FUNCTION_BLOCK FB_RecipeAnalogInputControlSequencer
VAR_INPUT
	rampTime: UINT;
END_VAR
VAR_IN_OUT
	rRecipe: ARRAY[1..GVL_IO.nNumController] OF REAL;
END_VAR
VAR
	i: INT;
END_VAR

FOR i:= 1 TO GVL_IO.nNumMFC DO
	GVL_IO.aController[i].input.restart := TRUE;
	GVL_IO.aController[i].input.rampTime := rampTime; 
	GVL_IO.aController[i].input.targetValue := rRecipe[i] / GVL_IO.aMaxValueController[i] * GVL_IO.EL3064MaxValueH;;
END_FOR

FOR i:= 1 TO GVL_IO.nNumFurnaceTemp DO
	GVL_IO.aController_TempContoller[i].input.restart := TRUE;
	GVL_IO.aController_TempContoller[i].input.rampTime := rampTime; 
	GVL_IO.aController_TempContoller[i].input.targetValue := rRecipe[i];
END_FOR

END_FUNCTION_BLOCK

(* stored: Version 1.1.0.1
   POU FB_RecipeAnalogInputControlSequencer: Id {e120b0c2-c4cf-40c9-aa7e-95c0a8deddb6}, SpecialFunc None *)
